ABB RobotStudio station: Project18.rsstnx

Station Project18 (saved by RobotStudio 22.3.10141.1)
Controller FYP_v00, task T_ROB1: task frame (RAPID world) sits at (0, 0, 1244) mm in the station
Controller FYP_v00
  mechanical unit ROB_1: CRB15000_5_95__02, 6 joints, base frame (0, 0, 0) mm
Layout (positions relative to the parent item):
  - CRB15000_5_95__02 [mechanism, from Robots\CRB15000_5_95__02.rslib] at (0, 0, 1244) mm; joint values [0, 1.0482, -0.5556, 0, 1.0786, 0] (rad or m)
  - Cell [graphiccomponentgroup] at (-115.88, -500, 0) mm, rotated rx 0 ry 0 rz 90 deg
    - Wagon [part] at (380, -350, 0) mm, size 1011.1 x 704 x 1240.9 mm
    - OmniCore_C30 [part, from %ABB.RobotStudio.Models.OmniCore%\OmniCore_C30.rslib] at (56.63, -527.32, 209.4) mm
  - Azure Kinect DK [part] at (793.5, 0.02, 1570.93) mm, rotated rx 179.98 ry 0 rz -90 deg, size 103 x 39 x 125.4 mm
  - Attacher [smart component]
      signals: DI pick, DI place
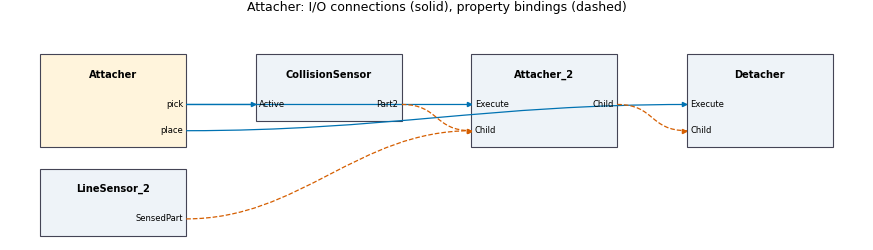
      connections:
        Attacher.pick -> CollisionSensor.Active
        Attacher.place -> Detacher.Execute
        Attacher.pick -> Attacher_2.Execute
        CollisionSensor.Part2 => Attacher_2.Child
        Attacher_2.Child => Detacher.Child
        LineSensor_2.SensedPart => Attacher_2.Child
    - Attacher_2 [smart component, from Components\Attacher.rslib]
        properties: Parent=SCHUNK-EGP-C-40_2; Flange=0; Child=(none); Mount=true; Offset=[0 0 0]; Orientation=[0 0 0]
    - Detacher [smart component, from Components\Detacher.rslib]
        properties: Child=(none); KeepPosition=true
    - LineSensor_2 [smart component, from Components\LineSensor.rslib] at (930.83, 0.02, 1504.26) mm, rotated rx 90.02 ry 0 rz 98.42 deg
        properties: Start=[-0.00441973579148422 -0.181951073673325 7.75364084550922E-05]; End=[0.00447229888785239 -0.18195131589354 0.00146616134082678]; Radius=0.009; SensedPart=(none); SensedPoint=[0 0 0]
      - _sensorPart_ [part], size 11.7 x 18 x 19.2 mm
  - Gripper [smart component]
      signals: DI open, DI close
      connections:
        Gripper.open -> PoseMover_2.Execute
        Gripper.close -> PoseMover.Execute
        Counter.Count => PoseMover.Pose
    - PoseMover [smart component, from Components\PoseMover.rslib]
        properties: Mechanism=SCHUNK-EGP-C-40_2; Pose=1; Duration=0.5
    - PoseMover_2 [smart component, from Components\PoseMover.rslib]
        properties: Mechanism=SCHUNK-EGP-C-40_2; Pose=2; Duration=0.5
  - SimulationEvents [smart component, from Components\SimulationEvents.rslib]
  - SCHUNK-EGP-C-40_2 [mechanism, from Components\SCHUNK-EGP-C-40_2.rslib] at (-1170.98, -0.09, 981.62) mm, rotated rx 0 ry 60.02 rz 0 deg; joint values [0.002, 0.002] (rad or m)
  - p2 [part] at (521.71, 181.62, 1254.32) mm, rotated rx -0.58 ry -0.65 rz 66.47 deg, size 50 x 20 x 20 mm
Attachment: Azure Kinect DK is attached to CRB15000_5_95__02 / Link5
Attachment: LineSensor_2 is attached to SCHUNK-EGP-C-40_2 / L1
Attachment: SCHUNK-EGP-C-40_2 is attached to CRB15000_5_95__02 / Link6
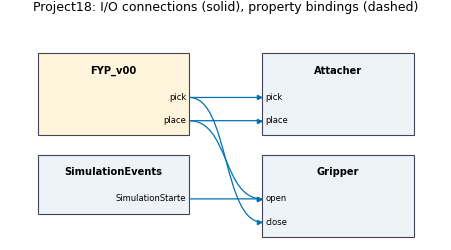
Station logic (signal -> signal, property => property):
  FYP_v00.pick -> Attacher.pick
  FYP_v00.place -> Gripper.open
  FYP_v00.pick -> Gripper.close
  FYP_v00.place -> Attacher.place
  SimulationEvents.SimulationStarted -> Gripper.open
Targets, tools, work objects and paths stored in the station, written as RAPID:
! task T_ROB1
MODULE MainModule
  CONST robtarget HOME_10:=[[550.168,0,522.381],[1,0,0,0],[0,0,0,0],[9E+09,9E+09,9E+09,9E+09,9E+09,9E+09]];
  CONST robtarget HOME_20:=[[736.426,0,665.702],[0.923879533,0,-0.382683432,0],[0,0,0,0],[9E+09,9E+09,9E+09,9E+09,9E+09,9E+09]];
  PROC calib_work()
    SetDO APAV_calibrateWorker,0;
    MoveL HOME_20,v1000,z100,Tooldata_1\WObj:=wobj0;
  ENDPROC
  PROC main()
    calib_rob;
    calib_work;
    pick_place;
    dataConversion;
    writeData;
    WaitTime 2;
  ENDPROC
  PROC calib_rob()
    SetDO APAV_calibrateRobot,0;
    MoveL HOME_10,v1000,z100,Tooldata_1\WObj:=wobj0;
  ENDPROC
  PROC pick_place()
  ENDPROC
  PROC dataConversion()
  ENDPROC
  PROC blocksDetection()
    SetDO APAV_piece_1,cubeM{4,4};
    SetDO APAV_piece_2,cubeM{4,4};
    SetDO APAV_piece_3,cubeM{4,4};
    SetDO APAV_piece_4,cubeM{4,4};
    SetDO APAV_piece_5,cubeM{4,4};
  ENDPROC
  PROC writeData()
  ENDPROC
ENDMODULE

! task T_ROB1
MODULE TorqueSensorCalib
  PROC TorqueSensorCal()
  ENDPROC
ENDMODULE

! task T_ROB1
MODULE CalibData
  PERS wobjdata Workobject_1:=[FALSE,TRUE,"",[[201.929992676,-200.789993286,3.49000001],[0.999960922,0.003150189,-0.006891656,0.004553765]],[[0,0,0],[1,0,0,0]]];
  PERS tooldata Tooldata_1:=[TRUE,[[0.19321156,0,204.571412367],[0.00026378,0.015111926,-0.999847707,-0.008724874]],[1,[0,0,1],[1,0,0,0],0,0,0]];
ENDMODULE

